// TIA Portal V17 export
// export: Created 2025-03-12T15:35:16.9898169Z, ExportSetting WithDefaults, DisplayName Totally Integrated Automation Portal, DisplayVersion V17 Update 8, DisplayName TIA Portal Openness, DisplayVersion V17 Update 8, DisplayName TIA Portal Version Control Interface, DisplayVersion V17, DisplayName SINAMICS Startdrive Advanced, DisplayVersion V17 SP2, DisplayName SINAMICS Startdrive G110M, G120, G120C, G120D, G120P, G115D, DisplayVersion V17 SP2, DisplayName SINAMICS Startdrive G130, G150, S120, S150, SINAMICS MV, S210, DisplayVersion V17 SP2, DisplayName STEP 7 Professional, DisplayVersion V17 Update 8, DisplayName SINUMERIK ONE STEP 7 Toolbox, DisplayVersion V17 Update 12, DisplayName SINUMERIK 840D sl STEP 7 Toolbox, DisplayVersion V17 Update 12, DisplayName STEP 7 Safety, DisplayVersion V17 Update 6, DisplayName WinCC Advanced, DisplayVersion V17 Update 8
DATA_BLOCK "DB2103_ELECTRICAL_CABINET"   // DB2103
{ S7_Optimized_Access := 'FALSE'; DB_Accessible_From_OPC_UA := 'FALSE' }
AUTHOR : ETXETAR
VERSION : 1.0
// stored: AutoNumber false, DBAccessibleFromOPCUA false, DBAccessibleFromWebserver true, IsOnlyStoredInLoadMemory false, IsWriteProtectedInAS false
   VAR RETAIN
      INPUT_MAIN_BREAKER : Bool;   // INPUT MAIN CABINET CIRCUIT BREAKER TRIPPED
      INPUT_AIR_UNIT_1_BREAKER : Bool;   // INPUT AIR UNIT 1 CRICUIT BREAKER TRIPPED
      INPUT_AIR_UNIT_2_BREAKER : Bool;   // INPUT AIR UNIT 2 CIRCUIT BREAKER TRIPPED
      INPUT_24VDC_BREAKER_1 : Bool;   // INPUT 24 VDC CIRCUIT BREAKER TRIPPED 1
      INPUT_24VDC_BREAKER_2 : Bool;   // INPUT 24 VDC CIRCUIT BREAKER TRIPPED 2
      INPUT_QFC03_BREAKER : Bool;   // INPUT QFC03 CIRCUIT BREAKER TRIPPED
      INPUT_SINAMICS_BREAKER : Bool;   // INPUT SINAMICS CIRCUIT BREAKER TRIPPED
      "INPUT_110/120/220/230VAC_BREAKER" : Bool;   // INPUT 110/120/220/230VAC CIRCUIT BREAKER TRIPPED
      INPUT_SINAMICS_BREAKER_1 : Bool;   // INPUT SINAMICS CIRCUIT BREAKER TRIPPED
      INPUT_CAB_LIGHT_BREAKER : Bool;   // INPUT CABINET LIGHT CIRCUIT BREAKER TRIPPED
      INPUT_SENTRON_PAC_BREAKER : Bool;   // INPUT SENTRON PAC CIRCUIT BREAKER TRIPPED
      INPUT_WATTMETER_BREAKER : Bool;   // INPUT WATTMETER CIRCUIT BREAKER TRIPPED
      INPUT_MAIN_SWITCH : Bool;   // INPUT MAIN SWITCH
      INPUT_PANEL_TEMPERATURE : Bool;   // INPUT PANEL TEMPERATURE
      INPUT_AIR_UNIT_1 : Bool;   // INPUT AIR UNIT 1
      INPUT_AIR_UNIT_2 : Bool;   // INPUT AIR UNIT 2
      INPUT_OVER_VOLTAGE : Bool;   // INPUT OVER VOLTAGE
      INPUT_POWER_SUPPLY : Bool;   // INPUT POWER SUPPLY
      INPUT_PS_24V_NOT_READY_DEV_1 : Bool;   // INPUT POWER SUPPLY 24V NOT READY DEVICE 1
      INPUT_PS_24V_NOT_READY_DEV_2 : Bool;   // INPUT POWER SUPPLY 24V NOT READY DEVICE 2
      INPUT_PS_24V_NOT_READY_DEV_3 : Bool;   // INPUT POWER SUPPLY 24V NOT READY DEVICE 3
      INPUT_PS_24V_NOT_READY_DEV_4 : Bool;   // INPUT POWER SUPPLY 24V NOT READY DEVICE 4
      INPUT_PS_24V_NOT_READY_DEV_5 : Bool;   // INPUT POWER SUPPLY 24V NOT READY DEVICE 5
      INPUT_PS_24V_NOT_READY_DEV_6 : Bool;   // INPUT POWER SUPPLY 24V NOT READY DEVICE 6
      INPUT_BATTERY_OK_SITOP_UPS500S : Bool;   // INPUT BATTERY OK SITOP UPS500S
      INPUT_BATTERY_ALARM_SITOP_UPS500S : Bool;   // INPUT BATTERY ALARM SITOP UPS500S
      INPUT_ETHERNET_SWITCH_1 : Bool;   // INPUT ETHERNET SWITCH 1
      INPUT_ETHERNET_SWITCH_2 : Bool;   // INPUT ETHERNET SWITCH 2
      INPUT_ETHERNET_SWITCH_3 : Bool;   // INPUT ETHERNET SWITCH 3
      INPUT_PROFINET_CTRL_UNIT_FAULT : Bool;   // INPUT PROFINET CONTROL UNIT FAULT
      INPUT_ETHERNET_SWITCH_4 : Bool;   // INPUT ETHERNET SWITCH 4
      INPUT_ELEC_CAB_DOOR_OPEN : Bool;   // INPUT ELECTRICAL CABINET DOOR OPEN
      INPUT_BATTERY_85_SITOP_UPS500S : Bool;   // INPUT BATTERY 85% SITOP UPS500S
      INPUT_PS_24V_BREAKER_DEV_1 : Bool;   // INPUT POWER SUPPLY 24V CIRCUIT BREAKER TRIPPED DEVICE 1
      INPUT_PS_24V_BREAKER_DEV_2 : Bool;   // INPUT POWER SUPPLY 24V CIRCUIT BREAKER TRIPPED DEVICE 2
      INPUT_PS_24V_BREAKER_DEV_3 : Bool;   // INPUT POWER SUPPLY 24V CIRCUIT BREAKER TRIPPED DEVICE 3
      INPUT_PS_24V_BREAKER_DEV_4 : Bool;   // INPUT POWER SUPPLY 24V CIRCUIT BREAKER TRIPPED DEVICE 4
      INPUT_LASER_BREAKER_U01 : Bool;   // INPUT LASER SOURCE UNIT 01 CIRCUIT BREAKER TRIPPED
      INPUT_LASER_BREAKER_U02 : Bool;   // INPUT LASER SOURCE UNIT 02 CIRCUIT BREAKER TRIPPED
      INPUT_OERLIKON_BREAKER_U01 : Bool;   // INPUT OERLIKON SOURCE UNIT 01 CIRCUIT BREAKER TRIPPED
      INPUT_OERLIKON_BREAKER_U02 : Bool;   // INPUT OERLIKON SOURCE UNIT 02 CIRCUIT BREAKER TRIPPED
      INPUT_HEATER_BREAKER : Bool;   // INPUT HEATER CIRCUIT BREAKER TRIPPED
      INPUT_STIRRER_BREAKER : Bool;   // INPUT STIRRER CIRCUIT BREAKER 2 TRIPPED
      INPUT_CONTROL_VOLTAGE_ON : Bool;   // INPUT CONTROL VOLTAGE ON
      INPUT_CONTROL_ON_ : Bool;   // INPUT CONTROL ON
      INPUT_CHILLER_BREAKER_1 : Bool;   // INPUT CHILLER CIRCUIT BREAKER 1 TRIPPED
      INPUT_CHILLER_BREAKER_2 : Bool;   // INPUT CHILLER CIRCUIT BREAKER 2 TRIPPED
      INPUT_CHILLER_BREAKER_3 : Bool;   // INPUT CHILLER CIRCUIT BREAKER 2 TRIPPED
      INPUT_HOPPERS_BREAKER : Bool;   // INPUT HOPPERS CIRCUIT BREAKER 2 TRIPPED
      INPUT_PC_CABINET_BREAKER : Bool;   // INPUT PC CABINET BREAKER TRIPPED
      INPUT_BREAKER_QFC40 : Bool;   // INPUT QFC40 BREAKER TRIPPED
      INPUT_BREAKER_QB02 : Bool;   // INPUT QB02 BREAKER TRIPPED
      INPUT_BREAKER_0FC30 : Bool;   // INPUT 0FC30 BREAKER TRIPPED
      INPUT_BREAKER_0FC20 : Bool;   // INPUT 0FC20 BREAKER TRIPPED
      INPUT_BREAKER_0FC21 : Bool;   // INPUT 0FC21 BREAKER TRIPPED
      INPUT_BREAKER_0FC22 : Bool;   // INPUT 0FC22 BREAKER TRIPPED
      INPUT_BREAKER_0FC23 : Bool;   // INPUT 0FC23 BREAKER TRIPPED
      INPUT_CIRCUIT_BREAKER_TRIPPED_LIGHT_STA_3 : Bool;   // INPUT CIRCUIT BREAKER TRIPPED LIGHT STATION 3
      INPUT_MIST_EXTRACTION_READY : Bool;   // INPUT MIST EXTRACTION READY
      INPUT_MIST_EXTRACTION_FAULT : Bool;   // INPUT MIST EXTRACTION FAULT
      INPUT_LASER_UNIT_01_OK : Bool;   // INPUT LASER UNIT 01 OK
      INPUT_LASER_UNIT_02_OK : Bool;   // INPUT LASER UNIT 02 OK
      INPUT_ROBOT_CELL_CIRCUIT_BREAKER : Bool;   // INPUT CELL CIRCUIT BREAKER TRIPPED
      INPUT_PILZ_ESTOP_OK : Bool;   // INPUT PILZ EMERGENCY STOP OK
      CONTROL_VOLTAGE_ON_ALARM : Bool;   // CONTROL VOLTAGE ON ALARM
      MAIN_BREAKER_TRIPPED_ALARM : Bool;   // MAIN CIRCUIT BREAKER TRIPPED ALARM
      AIR_UNIT_1_BREAKER_TRIPPED_ALARM : Bool;   // AIR UNIT 1 CIRCUIT BREAKER TRIPPED ALARM
      AIR_UNIT_2_BREAKER_TRIPPED_ALARM : Bool;   // AIR UNIT 2 CIRCUIT BREAKER TRIPPED ALARM
      "24VDC_BREAKER_TRIPPED_ALARM_1" : Bool;   // 24 VDC CIRCUIT BREAKER TRIPPED 1 ALARM
      "24VDC_BREAKER_TRIPPED_ALARM_2" : Bool;   // 24 VDC CIRCUIT BREAKER TRIPPED 2 ALARM
      QFC03_BREAKER_TRIPPED_ALARM : Bool;   // QFC03 CIRCUIT BREAKER TRIPPED ALARM
      SINAMICS_BREAKER_TRIPPED_ALARM : Bool;   // SINAMICS CIRCUIT BREAKER TRIPPED ALARM
      MAIN_SWITCH_ALARM : Bool;   // MAIN SWITCH ALARM
      PANEL_TEMPERATURE_ALARM : Bool;   // PANEL TEMPERATURE ALARM
      AIR_UNIT_ALARM_1 : Bool;   // AIR UNIT 1 ALARM
      AIR_UNIT_ALARM_2 : Bool;   // AIR UNIT 2 ALARM
      OVER_VOLTAGE_ALARM : Bool;   // OVER VOLTAGE ALARM
      POWER_SUPPLY_ALARM : Bool;   // POWER SUPPLY ALARM
      PS_24V_NOT_READY_DEV_ALARM_1 : Bool;   // POWER SUPPLY 24V NOT READY DEVICE 1 ALARM
      PS_24V_NOT_READY_DEV_ALARM_2 : Bool;   // POWER SUPPLY 24V NOT READY DEVICE 2 ALARM
      PS_24V_NOT_READY_DEV_ALARM_3 : Bool;   // POWER SUPPLY 24V NOT READY DEVICE 3 ALARM
      PS_24V_NOT_READY_DEV_ALARM_4 : Bool;   // POWER SUPPLY 24V NOT READY DEVICE 4 ALARM
      PS_24V_NOT_READY_DEV_ALARM_5 : Bool;   // POWER SUPPLY 24V NOT READY DEVICE 5 ALARM
      PS_24V_NOT_READY_DEV_ALARM_6 : Bool;   // POWER SUPPLY 24V NOT READY DEVICE 6 ALARM
      BATTERY_OK_SITOP_UPS500S_ALARM : Bool;   // BATTERY OK SITOP UPS500S ALARM
      BATTERY_ALARM_SITOP_UPS500S : Bool;   // BATTERY ALARM SITOP UPS500S ALARM
      ETHERNET_SWITCH_1_ALARM : Bool;   // ETHERNET SWITCH 1 ALARM
      ETHERNET_SWITCH_2_ALARM : Bool;   // ETHERNET SWITCH 2 ALARM
      ETHERNET_SWITCH_3_ALARM : Bool;   // ETHERNET SWITCH 3 ALARM
      PROFINET_CTRL_UNIT_FAULT_ALARM : Bool;   // PROFINET CONTROL UNIT FAULT ALARM
      ETHERNET_SWITCH_4_ALARM : Bool;   // ETHERNET SWITCH 4 ALARM
      PS_24V_BREAKER_TRIPPED_ALARM_DEV_1 : Bool;   // POWER SUPPLY 24V CIRCUIT BREAKER TRIPPED DEVICE 1 ALARM
      PS_24V_BREAKER_TRIPPED_ALARM_DEV_2 : Bool;   // POWER SUPPLY 24V CIRCUIT BREAKER TRIPPED DEVICE 2 ALARM
      PS_24V_BREAKER_TRIPPED_ALARM_DEV_3 : Bool;   // POWER SUPPLY 24V CIRCUIT BREAKER TRIPPED DEVICE 3 ALARM
      PS_24V_BREAKER_TRIPPED_ALARM_DEV_4 : Bool;   // POWER SUPPLY 24V CIRCUIT BREAKER TRIPPED DEVICE 4 ALARM
      SINAMICS_BREAKER_ALARM : Bool;   // SINAMICS CIRCUIT BREAKER TRIPPED ALARM
      LASER_BREAKER_U01_ALARM : Bool;   // ALARM LASER SOURCE UNIT 01 CIRCUIT BREAKER TRIPPED
      LASER_BREAKER_U02_ALARM : Bool;   // ALARM LASER SOURCE UNIT 02 CIRCUIT BREAKER TRIPPED
      OERLIKON_BREAKER_U01_ALARM : Bool;   // ALARM OERLIKON SOURCE UNIT 01 CIRCUIT BREAKER TRIPPED
      OERLIKON_BREAKER_U02_ALARM : Bool;   // ALARM OERLIKON SOURCE UNIT 02 CIRCUIT BREAKER TRIPPED
      HEATER_BREAKER_ALARM : Bool;   // ALARM HEATER CIRCUIT BREAKER TRIPPED
      STIRRER_BREAKER_ALARM : Bool;   // ALARM STIRRER CIRCUIT BREAKER TRIPPED
      CHILLER_1_BREAKER_ALARM : Bool;   // ALARM CHILLER CIRCUIT BREAKER TRIPPED
      CHILLER_2_BREAKER_ALARM : Bool;   // ALARM CHILLER CIRCUIT BREAKER TRIPPED
      HOPPERS_BREAKER_ALARM : Bool;   // ALARM HOPPERS CIRCUIT BREAKER TRIPPED
      ROBOT_CELL_BREAKER_ALARM : Bool;   // ALARM ROBOT CELL CIRCUIT BREAKER TRIPPED
      QFC40_BREAKER_ALARM : Bool;   // ALARM QFC40 CIRCUIT BREAKER TRIPPED
      QB02_BREAKER_ALARM : Bool;   // ALARM QB02 CIRCUIT BREAKER TRIPPED
      "0F06_BREAKER_ALARM" : Bool;   // ALARM 0F06 CIRCUIT BREAKER TRIPPED
      CIRCUIT_BREAKER_TRIPPED_LIGHT_STA_3_ALARM : Bool;   // ALARM CIRCUIT BREAKER TRIPPED LIGHT STATION 3
      MIST_EXTRACTION_READY_ALARM : Bool;   // MIST EXTRACTION READY ALARM
      MIST_EXTRACTION_FAULT_ALARM : Bool;   // MIST EXTRACTION FAULT ALARM
      LASER_UNIT_01_OK_ALARM : Bool;   // LASER UNIT 01 OK ALARM
      LASER_UNIT_02_OK_ALARM : Bool;   // LASER UNIT 02 OK ALARM
      "110/120/220/230VAC_BREAKER_TRIPPED_WARNING" : Bool;   // 110/120/220/230VAC CIRCUIT BREAKER TRIPPED WARNING
      CAB_LIGHT_BREAKER_TRIPPED_WARNING : Bool;   // CABINET LIGHT CIRCUIT BREAKER TRIPPED WARNING
      SENTRON_PAC_BREAKER_TRIPPED_WARNING : Bool;   // SENTRON PAC CIRCUIT BREAKER TRIPPED WARNING
      WATTMETER_BREAKER_TRIPPED_WARNING : Bool;   // JIB CRANE CIRCUIT BREAKER TRIPPED WARNING
      ELEC_CAB_DOOR_OPEN_WARNING : Bool;   // ELECTRICAL CABINET DOOR OPEN WARNING
      BATTERY_85_SITOP_UPS500S_WARNING : Bool;   // BATTERY 85% SITOP UPS500S WARNING
      "0FC20_BREAKER_WARNING" : Bool;   // 0FC20 CIRCUIT BREAKER TRIPPED WARNING
      "0FC21_BREAKER_WARNING" : Bool;   // 0FC21 CIRCUIT BREAKER TRIPPED WARNING
      "0FC22_BREAKER_WARNING" : Bool;   // 0FC22 CIRCUIT BREAKER TRIPPED WARNING
      "0FC23_BREAKER_WARNING" : Bool;   // 0FC23 CIRCUIT BREAKER TRIPPED WARNING
      PILZ_ESTOP_OK_WARNING : Bool;   // PILZ EMERGENCY STOP OK ALARM
      ANY_ACTIVE_ALARM : Bool;   // ANY ACTIVE ALARM
      IS_ALARMS : Bool;   // IMMEDIATE STOP ALARMS
      SEOC_ALARMS : Bool;   // STOP END OF CYCLE ALARMS
      WARNINGS : Bool;   // WARNINGS
      WARNINGS_GONE : Bool;   // WARNINGS GONE
      TIMER_SITOP_BATTERY { S7_SetPoint := 'True'} : TON_TIME;   // SITOP BATTERY TIMER
   END_VAR
BEGIN
   TIMER_SITOP_BATTERY.PT := T#5s;
END_DATA_BLOCK
